(* IEC 61131-3 sources: Lasal/CPU_5344_V01/Class/statusSafety, 1 file *)

(* ---- statusSafety.st ---- *)
(*!
<Class
	Name               = "statusSafety"
	Revision           = "0.0"
	RealtimeTask       = "false"
	CyclicTask         = "false"
	BackgroundTask     = "false"
	Sigmatek           = "false"
	OSInterface        = "false"
	HighPriority       = "false"
	Automatic          = "false"
	UpdateMode         = "Prescan"
	SharedCommandTable = "true"
	Objectsize         = "(360,720)">
	<Channels>
		<Server Name="ClassSvr" Visualized="false" Initialize="false" WriteProtected="true" Retentive="false"/>
		<Server Name="stsInputs1" Visualized="true" Initialize="false" WriteProtected="false" Retentive="false"/>
		<Server Name="stsInputs10" Visualized="true" Initialize="false" WriteProtected="false" Retentive="false"/>
		<Server Name="stsInputs2" Visualized="true" Initialize="false" WriteProtected="false" Retentive="false"/>
		<Server Name="stsInputs3" Visualized="true" Initialize="false" WriteProtected="false" Retentive="false"/>
		<Server Name="stsInputs4" Visualized="true" Initialize="false" WriteProtected="false" Retentive="false"/>
		<Server Name="stsInputs5" Visualized="true" Initialize="false" WriteProtected="false" Retentive="false"/>
		<Server Name="stsInputs6" Visualized="true" Initialize="false" WriteProtected="false" Retentive="false"/>
		<Server Name="stsInputs7" Visualized="true" Initialize="false" WriteProtected="false" Retentive="false"/>
		<Server Name="stsInputs8" Visualized="true" Initialize="false" WriteProtected="false" Retentive="false"/>
		<Server Name="stsInputs9" Visualized="true" Initialize="false" WriteProtected="false" Retentive="false"/>
	</Channels>
</Class>
*)
statusSafety : CLASS
  //Servers:
	ClassSvr 	: SvrChCmd_DINT;
	stsInputs1 	: SvrCh_DINT;
	stsInputs2 	: SvrCh_DINT;
	stsInputs3 	: SvrCh_DINT;
	stsInputs4 	: SvrCh_DINT;
	stsInputs5 	: SvrCh_DINT;
	stsInputs6 	: SvrCh_DINT;
	stsInputs7 	: SvrCh_DINT;
	stsInputs8 	: SvrCh_DINT;
	stsInputs9 	: SvrCh_DINT;
	stsInputs10 	: SvrCh_DINT;
  //Clients:
  //Variables:
  //Functions:
  //Tables:
	FUNCTION @STD
		VAR_OUTPUT
			ret_code	: CONFSTATES;
		END_VAR;
	FUNCTION GLOBAL TAB @CT_;
END_CLASS;
